// TIA Portal project "DIGITAL ASSEMBLER _Sequential" (V16)
// Vorlageprojekt für das Buch mit Zielsystem S7-1200

(* hardware
DEVICE "S7-1200-Station_1"  S7-1200 Station
   slot 0: "Baugruppenträger_0"  Rack  V1.0
   slot 1: "PLC_1"  CPU 1211C DC/DC/DC  6ES7 211-1AE40-0XB0  V4.1
DEVICE "S7300/ET200M station_1"  S7-300 station
   slot 0: "IO device_1"  IM 153-4 PN  6ES7 153-4BA00-0XB0  V4.0
   slot 0: "Rail_0"  Rail  6ES7 390-1***0-0AA0
   slot 1: "DI 16x24VDC_1"  DI16 x 24VDC  6ES7 321-1BH02-0AA0
   slot 2: "DO 16x24VDC/0.5A_1"  DO16 x 24VDC / 0.5A  6ES7 322-1BH01-0AA0
*)

// ===== PLC "PLC_1"  CPU 1211C DC/DC/DC =====

VAR_GLOBAL   // PLC tag table "Standard-Variablentabelle"
   "counter" AT %QD30 : UDInt;
   "stop light" AT %Q2.3 : Bool;
   "reset light'" AT %Q2.2 : Bool;
   "start light" AT %Q2.1 : Bool;
   "pos rise base" AT %Q2.0 : Bool;
   "clamp base" AT %Q1.7 : Bool;
   "pos rise lid" AT %Q1.6 : Bool;
   "base conveyor" AT %Q1.5 : Bool;
   "clamp lid" AT %Q1.4 : Bool;
   "lids conveyor" AT %Q1.3 : Bool;
   "grab" AT %Q1.2 : Bool;
   "move z" AT %Q1.1 : Bool;
   "move x" AT %Q1.0 : Bool;
   "auto" AT %I2.6 : Bool;
   "emergency stop" AT %I2.5 : Bool;
   "stop" AT %I2.4 : Bool;
   "reset" AT %I2.3 : Bool;
   "start" AT %I2.2 : Bool;
   "part leaving" AT %I2.1 : Bool;
   "pos at limit base" AT %I2.0 : Bool;
   "base clamped" AT %I1.7 : Bool;
   "base at place" AT %I1.6 : Bool;
   "pos at limit lid" AT %I1.5 : Bool;
   "lid clamped" AT %I1.4 : Bool;
   "lid at place" AT %I1.3 : Bool;
   "item detected" AT %I1.2 : Bool;
   "moving z" AT %I1.1 : Bool;
   "moving x" AT %I1.0 : Bool;
   "Manual" AT %I2.7 : Bool;
   "Memory_for_Steps" AT %M0.1 : Bool;
   "Start_FC_one_time" AT %M0.2 : Bool;
   "Tag_1" AT %M0.3 : Bool;
   "Tag_2" AT %M0.4 : Bool;
   "Tag_3" AT %M0.5 : Bool;
   "Tag_4" AT %M0.7 : Bool;
   "Tag_5" AT %M2.7 : Bool;
   "cycle_complete" AT %M3.0 : Bool;
   "Tag_6" AT %M4.1 : Bool;
   "Tag_7" AT %M4.2 : Bool;
   "Tag_8" AT %M5.0 : Bool;
   "Tag_9" AT %M5.1 : Bool;
   "Tag_10" AT %M5.2 : Bool;
   "Tag_11" AT %M5.3 : Bool;
   "Tag_12" AT %M5.4 : Bool;
   "Tag_13" AT %QW30 : Int;
END_VAR

DATA_BLOCK "modes"   // DB1
{ S7_Optimized_Access := 'FALSE' }
VERSION : 0.1
   VAR
      "Reset Mode" : Bool;
      "Manual Mode" : Bool;
      "Auto Mode" : Bool;
   END_VAR
BEGIN
END_DATA_BLOCK

DATA_BLOCK "Step_Data"   // DB2
{ S7_Optimized_Access := 'TRUE' }
VERSION : 0.1
   VAR
      Start_Lids_Conveyor : Bool;   // trun on lids conveyor
      Start_Base_conveyor : Bool;   // turn on base conveyor
      Start_Clamp_Lid : Bool;
      Start_Clamp_Base : Bool;
      Extend_Z_Axis : Bool;
      Extend_x_Axis : Bool;
      Start_Grap : Bool;
      Pose_raise_Base : Bool;
      Every_thing_AT_home : Bool;
   END_VAR
BEGIN
END_DATA_BLOCK

DATA_BLOCK "Steps"   // DB3
{ S7_Optimized_Access := 'TRUE' }
VERSION : 0.1
   VAR
      Current_step : Int;
   END_VAR
BEGIN
END_DATA_BLOCK

// folder: System blocks/Program resources

DATA_BLOCK "IEC_Counter_0_DB"   // DB4
{ S7_Optimized_Access := 'TRUE' }
AUTHOR : Simatic
FAMILY : IEC
NAME : CNTR
VERSION : 1.0
// stored: InstanceOfName IEC_COUNTER
"IEC_COUNTER"
BEGIN
END_DATA_BLOCK

// folder: (top level)

FUNCTION "Operating Mode" : Void   // FC1, LAD
{ S7_Optimized_Access := 'TRUE' }
VERSION : 0.1
   VAR_TEMP   // added for the SCL form of the ladder/FBD networks
      _w1 : Bool;
      _w2 : Bool;
   END_VAR
BEGIN

REGION Network 1
   // manual
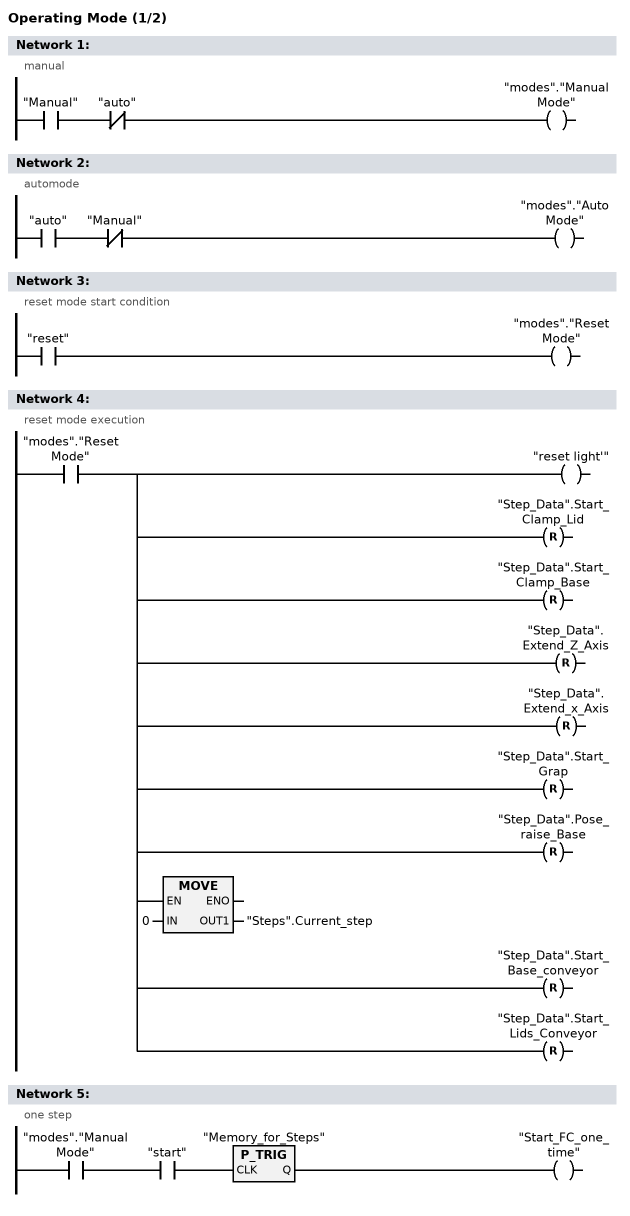
   RUNG wire#powerrail
      Contact( "Manual" )
      I_Contact( "auto" )
      Coil( "modes"."Manual Mode" )
   END_RUNG
   // the same network as SCL:
   "modes"."Manual Mode" := "Manual" AND NOT "auto";
END_REGION

REGION Network 2
   // automode
   RUNG wire#powerrail
      Contact( "auto" )
      I_Contact( "Manual" )
      Coil( "modes"."Auto Mode" )
   END_RUNG
   // the same network as SCL:
   "modes"."Auto Mode" := "auto" AND NOT "Manual";
END_REGION

REGION Network 3
   // reset mode start condition
   RUNG wire#powerrail
      Contact( "reset" )
      Coil( "modes"."Reset Mode" )
   END_RUNG
   // the same network as SCL:
   "modes"."Reset Mode" := "reset";
END_REGION

REGION Network 4
   // reset mode execution
   RUNG wire#powerrail
      Contact( "modes"."Reset Mode" )
      wire#w1
      Coil( "reset light'" )
   END_RUNG
   RUNG wire#w1
      R_Coil( "Step_Data".Start_Clamp_Lid )
   END_RUNG
   RUNG wire#w1
      R_Coil( "Step_Data".Start_Clamp_Base )
   END_RUNG
   RUNG wire#w1
      R_Coil( "Step_Data".Extend_Z_Axis )
   END_RUNG
   RUNG wire#w1
      R_Coil( "Step_Data".Extend_x_Axis )
   END_RUNG
   RUNG wire#w1
      R_Coil( "Step_Data".Start_Grap )
   END_RUNG
   RUNG wire#w1
      R_Coil( "Step_Data".Pose_raise_Base )
   END_RUNG
   RUNG wire#w1
      Move(in := 0, out1 => "Steps".Current_step)
   END_RUNG
   RUNG wire#w1
      R_Coil( "Step_Data".Start_Base_conveyor )
   END_RUNG
   RUNG wire#w1
      R_Coil( "Step_Data".Start_Lids_Conveyor )
   END_RUNG
   // the same network as SCL:
   "reset light'" := "modes"."Reset Mode";
   IF "modes"."Reset Mode" THEN
       "Step_Data".Start_Clamp_Lid := FALSE;
       "Step_Data".Start_Clamp_Base := FALSE;
       "Step_Data".Extend_Z_Axis := FALSE;
       "Step_Data".Extend_x_Axis := FALSE;
       "Step_Data".Start_Grap := FALSE;
       "Step_Data".Pose_raise_Base := FALSE;
       "Steps".Current_step := 0;
       "Step_Data".Start_Base_conveyor := FALSE;
       "Step_Data".Start_Lids_Conveyor := FALSE;
   END_IF;
END_REGION

REGION Network 5
   // one step
   RUNG wire#powerrail
      Contact( "modes"."Manual Mode" )
      Contact( "start" )
      P_Trig( "Memory_for_Steps" )
      Coil( "Start_FC_one_time" )
   END_RUNG
   // the same network as SCL:
   #_w1 := "modes"."Manual Mode" AND "start";
   #_w2 := #_w1 AND NOT "Memory_for_Steps";   // rising edge
   "Memory_for_Steps" := #_w1;
   "Start_FC_one_time" := #_w2;
END_REGION

REGION Network 6
   // make sure envery thing is reseted before starting
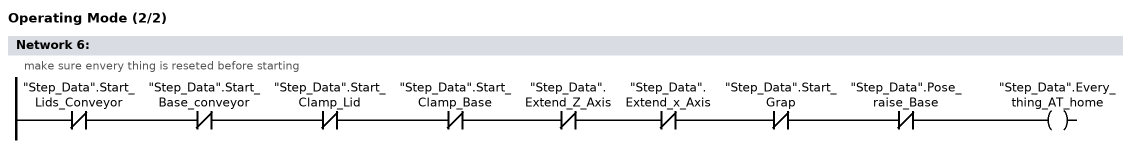
   RUNG wire#powerrail
      I_Contact( "Step_Data".Start_Lids_Conveyor )
      I_Contact( "Step_Data".Start_Base_conveyor )
      I_Contact( "Step_Data".Start_Clamp_Lid )
      I_Contact( "Step_Data".Start_Clamp_Base )
      I_Contact( "Step_Data".Extend_Z_Axis )
      I_Contact( "Step_Data".Extend_x_Axis )
      I_Contact( "Step_Data".Start_Grap )
      I_Contact( "Step_Data".Pose_raise_Base )
      Coil( "Step_Data".Every_thing_AT_home )
   END_RUNG
   // the same network as SCL:
   "Step_Data".Every_thing_AT_home := NOT "Step_Data".Start_Lids_Conveyor AND NOT "Step_Data".Start_Base_conveyor AND NOT "Step_Data".Start_Clamp_Lid AND NOT "Step_Data".Start_Clamp_Base AND NOT "Step_Data".Extend_Z_Axis AND NOT "Step_Data".Extend_x_Axis AND NOT "Step_Data".Start_Grap AND NOT "Step_Data".Pose_raise_Base;
END_REGION
END_FUNCTION

FUNCTION "Step_definition" : Void   // FC2, LAD
{ S7_Optimized_Access := 'TRUE' }
VERSION : 0.1
   VAR_TEMP   // added for the SCL form of the ladder/FBD networks
      _w1 : Bool;
   END_VAR
BEGIN

REGION Network 1: start lids conveyor till lid at place
   // start pressed  and every thing at home
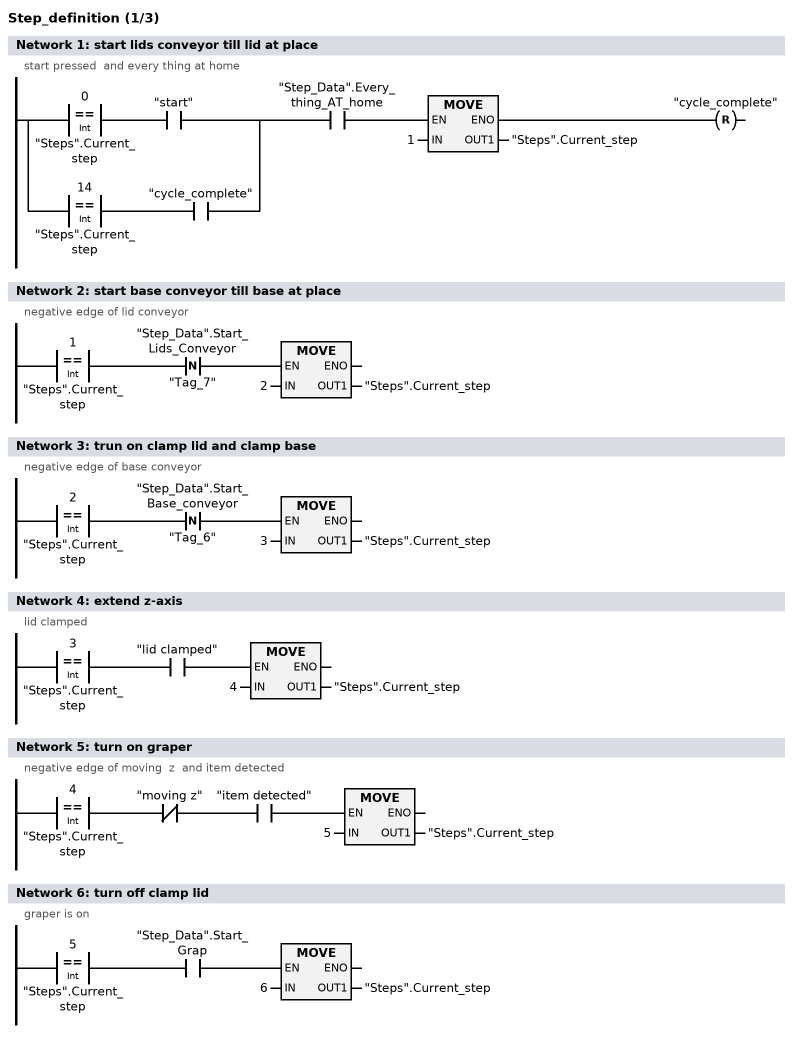
   RUNG wire#powerrail
      { S7_Templates := "SrcType := Int" } EQ_Contact(in1 := 0, in2 := "Steps".Current_step)
      Contact( "start" )
      wire#w1
      Contact( "Step_Data".Every_thing_AT_home )
      Move(in := 1, out1 => "Steps".Current_step)
      R_Coil( "cycle_complete" )
   END_RUNG
   RUNG wire#powerrail
      { S7_Templates := "SrcType := Int" } EQ_Contact(in1 := 14, in2 := "Steps".Current_step)
      Contact( "cycle_complete" )
   END_RUNG wire#w1
   // the same network as SCL:
   #_w1 := (((0 = "Steps".Current_step) AND "start") OR ((14 = "Steps".Current_step) AND "cycle_complete")) AND "Step_Data".Every_thing_AT_home;
   IF #_w1 THEN
       "Steps".Current_step := 1;
       "cycle_complete" := FALSE;
   END_IF;
END_REGION

REGION Network 2: start base conveyor till base at place
   // negative edge of lid conveyor
   RUNG wire#powerrail
      { S7_Templates := "SrcType := Int" } EQ_Contact(in1 := 1, in2 := "Steps".Current_step)
      N_Contact(operand := "Step_Data".Start_Lids_Conveyor, bit := "Tag_7")
      Move(in := 2, out1 => "Steps".Current_step)
   END_RUNG
   // the same network as SCL:
   #_w1 := (1 = "Steps".Current_step) AND NOT "Step_Data".Start_Lids_Conveyor AND "Tag_7";   // falling edge of "Step_Data".Start_Lids_Conveyor
   "Tag_7" := "Step_Data".Start_Lids_Conveyor;
   IF #_w1 THEN "Steps".Current_step := 2; END_IF;
END_REGION

REGION Network 3: trun on clamp lid and clamp base
   // negative edge of base conveyor
   RUNG wire#powerrail
      { S7_Templates := "SrcType := Int" } EQ_Contact(in1 := 2, in2 := "Steps".Current_step)
      N_Contact(operand := "Step_Data".Start_Base_conveyor, bit := "Tag_6")
      Move(in := 3, out1 => "Steps".Current_step)
   END_RUNG
   // the same network as SCL:
   #_w1 := (2 = "Steps".Current_step) AND NOT "Step_Data".Start_Base_conveyor AND "Tag_6";   // falling edge of "Step_Data".Start_Base_conveyor
   "Tag_6" := "Step_Data".Start_Base_conveyor;
   IF #_w1 THEN "Steps".Current_step := 3; END_IF;
END_REGION

REGION Network 4: extend z-axis
   // lid clamped
   RUNG wire#powerrail
      { S7_Templates := "SrcType := Int" } EQ_Contact(in1 := 3, in2 := "Steps".Current_step)
      Contact( "lid clamped" )
      Move(in := 4, out1 => "Steps".Current_step)
   END_RUNG
   // the same network as SCL:
   IF (3 = "Steps".Current_step) AND "lid clamped" THEN "Steps".Current_step := 4; END_IF;
END_REGION

REGION Network 5: turn on graper
   // negative edge of moving  z  and item detected
   RUNG wire#powerrail
      { S7_Templates := "SrcType := Int" } EQ_Contact(in1 := 4, in2 := "Steps".Current_step)
      I_Contact( "moving z" )
      Contact( "item detected" )
      Move(in := 5, out1 => "Steps".Current_step)
   END_RUNG
   // the same network as SCL:
   IF (4 = "Steps".Current_step) AND NOT "moving z" AND "item detected" THEN
       "Steps".Current_step := 5;
   END_IF;
END_REGION

REGION Network 6: turn off clamp lid
   // graper is on
   RUNG wire#powerrail
      { S7_Templates := "SrcType := Int" } EQ_Contact(in1 := 5, in2 := "Steps".Current_step)
      Contact( "Step_Data".Start_Grap )
      Move(in := 6, out1 => "Steps".Current_step)
   END_RUNG
   // the same network as SCL:
   IF (5 = "Steps".Current_step) AND "Step_Data".Start_Grap THEN "Steps".Current_step := 6; END_IF;
END_REGION

REGION Network 7: retract z-axis
   // lid clamped off
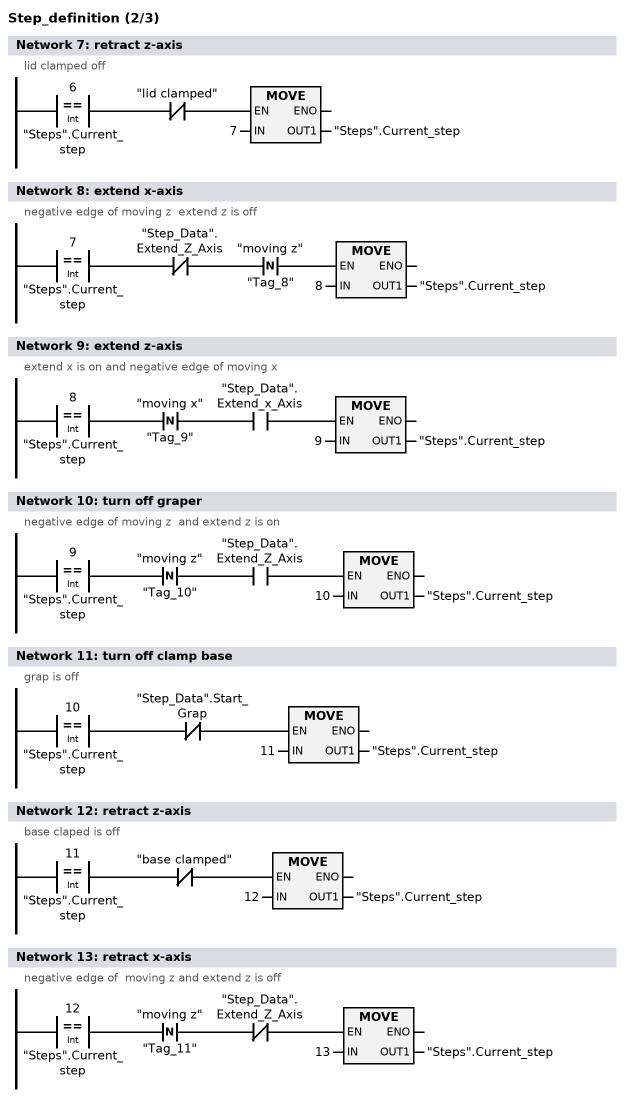
   RUNG wire#powerrail
      { S7_Templates := "SrcType := Int" } EQ_Contact(in1 := 6, in2 := "Steps".Current_step)
      I_Contact( "lid clamped" )
      Move(in := 7, out1 => "Steps".Current_step)
   END_RUNG
   // the same network as SCL:
   IF (6 = "Steps".Current_step) AND NOT "lid clamped" THEN "Steps".Current_step := 7; END_IF;
END_REGION

REGION Network 8: extend x-axis
   // negative edge of moving z  extend z is off
   RUNG wire#powerrail
      { S7_Templates := "SrcType := Int" } EQ_Contact(in1 := 7, in2 := "Steps".Current_step)
      I_Contact( "Step_Data".Extend_Z_Axis )
      N_Contact(operand := "moving z", bit := "Tag_8")
      Move(in := 8, out1 => "Steps".Current_step)
   END_RUNG
   // the same network as SCL:
   #_w1 := (7 = "Steps".Current_step) AND NOT "Step_Data".Extend_Z_Axis AND NOT "moving z" AND "Tag_8";   // falling edge of "moving z"
   "Tag_8" := "moving z";
   IF #_w1 THEN "Steps".Current_step := 8; END_IF;
END_REGION

REGION Network 9: extend z-axis
   // extend x is on and negative edge of moving x
   RUNG wire#powerrail
      { S7_Templates := "SrcType := Int" } EQ_Contact(in1 := 8, in2 := "Steps".Current_step)
      N_Contact(operand := "moving x", bit := "Tag_9")
      Contact( "Step_Data".Extend_x_Axis )
      Move(in := 9, out1 => "Steps".Current_step)
   END_RUNG
   // the same network as SCL:
   #_w1 := (8 = "Steps".Current_step) AND NOT "moving x" AND "Tag_9";   // falling edge of "moving x"
   "Tag_9" := "moving x";
   IF #_w1 AND "Step_Data".Extend_x_Axis THEN "Steps".Current_step := 9; END_IF;
END_REGION

REGION Network 10: turn off graper
   // negative edge of moving z  and extend z is on
   RUNG wire#powerrail
      { S7_Templates := "SrcType := Int" } EQ_Contact(in1 := 9, in2 := "Steps".Current_step)
      N_Contact(operand := "moving z", bit := "Tag_10")
      Contact( "Step_Data".Extend_Z_Axis )
      Move(in := 10, out1 => "Steps".Current_step)
   END_RUNG
   // the same network as SCL:
   #_w1 := (9 = "Steps".Current_step) AND NOT "moving z" AND "Tag_10";   // falling edge of "moving z"
   "Tag_10" := "moving z";
   IF #_w1 AND "Step_Data".Extend_Z_Axis THEN "Steps".Current_step := 10; END_IF;
END_REGION

REGION Network 11: turn off clamp base
   // grap is off
   RUNG wire#powerrail
      { S7_Templates := "SrcType := Int" } EQ_Contact(in1 := 10, in2 := "Steps".Current_step)
      I_Contact( "Step_Data".Start_Grap )
      Move(in := 11, out1 => "Steps".Current_step)
   END_RUNG
   // the same network as SCL:
   IF (10 = "Steps".Current_step) AND NOT "Step_Data".Start_Grap THEN "Steps".Current_step := 11; END_IF;
END_REGION

REGION Network 12: retract z-axis
   // base claped is off
   RUNG wire#powerrail
      { S7_Templates := "SrcType := Int" } EQ_Contact(in1 := 11, in2 := "Steps".Current_step)
      I_Contact( "base clamped" )
      Move(in := 12, out1 => "Steps".Current_step)
   END_RUNG
   // the same network as SCL:
   IF (11 = "Steps".Current_step) AND NOT "base clamped" THEN "Steps".Current_step := 12; END_IF;
END_REGION

REGION Network 13: retract x-axis
   // negative edge of  moving z and extend z is off
   RUNG wire#powerrail
      { S7_Templates := "SrcType := Int" } EQ_Contact(in1 := 12, in2 := "Steps".Current_step)
      N_Contact(operand := "moving z", bit := "Tag_11")
      I_Contact( "Step_Data".Extend_Z_Axis )
      Move(in := 13, out1 => "Steps".Current_step)
   END_RUNG
   // the same network as SCL:
   #_w1 := (12 = "Steps".Current_step) AND NOT "moving z" AND "Tag_11";   // falling edge of "moving z"
   "Tag_11" := "moving z";
   IF #_w1 AND NOT "Step_Data".Extend_Z_Axis THEN "Steps".Current_step := 13; END_IF;
END_REGION

REGION Network 14: pose raise(base on)- base conveyor on till part leaving and counter +1 after part leaving
   // negative edge of  moving x and extend x is off
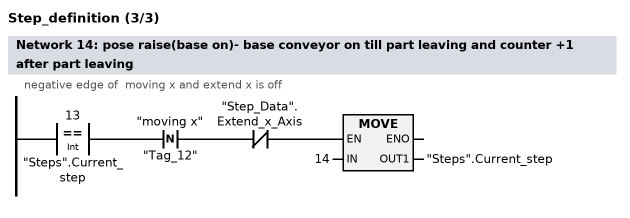
   RUNG wire#powerrail
      { S7_Templates := "SrcType := Int" } EQ_Contact(in1 := 13, in2 := "Steps".Current_step)
      N_Contact(operand := "moving x", bit := "Tag_12")
      I_Contact( "Step_Data".Extend_x_Axis )
      Move(in := 14, out1 => "Steps".Current_step)
   END_RUNG
   // the same network as SCL:
   #_w1 := (13 = "Steps".Current_step) AND NOT "moving x" AND "Tag_12";   // falling edge of "moving x"
   "Tag_12" := "moving x";
   IF #_w1 AND NOT "Step_Data".Extend_x_Axis THEN "Steps".Current_step := 14; END_IF;
END_REGION
END_FUNCTION

FUNCTION "Step_Execution" : Void   // FC3, LAD
{ S7_Optimized_Access := 'TRUE' }
VERSION : 0.1
   VAR_TEMP   // added for the SCL form of the ladder/FBD networks
      _w1 : Bool;
      _w2 : Bool;
   END_VAR
BEGIN

REGION Network 1: trun on lids conveyor
   // start lids conveyor till lid at place
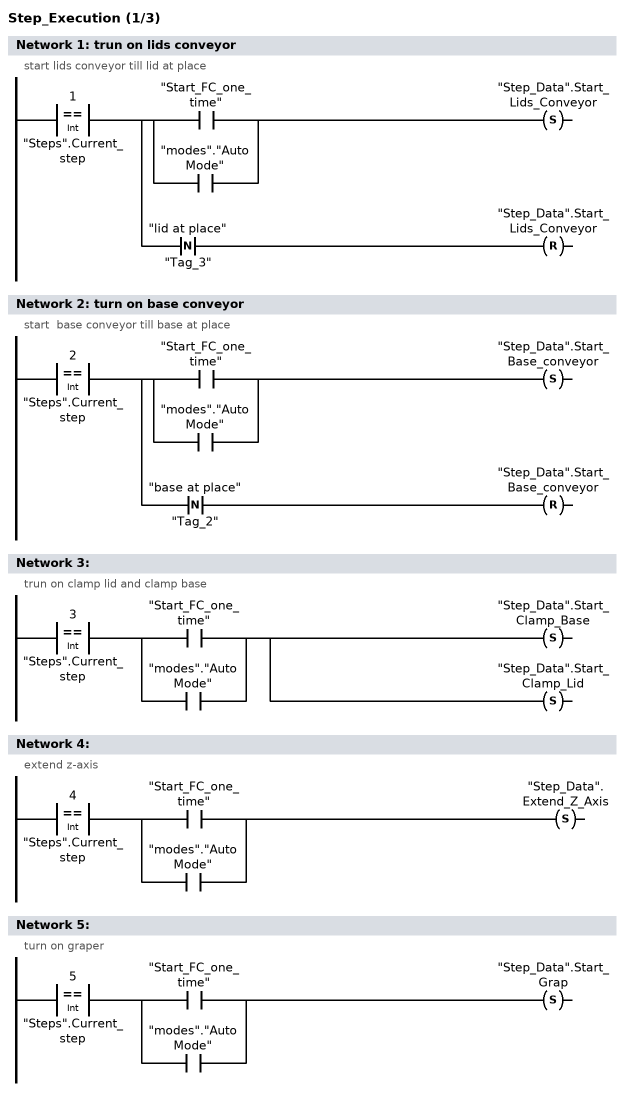
   RUNG wire#powerrail
      { S7_Templates := "SrcType := Int" } EQ_Contact(in1 := 1, in2 := "Steps".Current_step)
      wire#w1
      Contact( "Start_FC_one_time" )
      wire#w2
      S_Coil( "Step_Data".Start_Lids_Conveyor )
   END_RUNG
   RUNG wire#w1
      Contact( "modes"."Auto Mode" )
   END_RUNG wire#w2
   RUNG wire#w1
      N_Contact(operand := "lid at place", bit := "Tag_3")
      R_Coil( "Step_Data".Start_Lids_Conveyor )
   END_RUNG
   // the same network as SCL:
   #_w1 := 1 = "Steps".Current_step;
   IF #_w1 AND ("Start_FC_one_time" OR "modes"."Auto Mode") THEN
       "Step_Data".Start_Lids_Conveyor := TRUE;
   END_IF;
   #_w2 := #_w1 AND NOT "lid at place" AND "Tag_3";   // falling edge of "lid at place"
   "Tag_3" := "lid at place";
   IF #_w2 THEN "Step_Data".Start_Lids_Conveyor := FALSE; END_IF;
END_REGION

REGION Network 2: turn on base conveyor
   // start  base conveyor till base at place
   RUNG wire#powerrail
      { S7_Templates := "SrcType := Int" } EQ_Contact(in1 := 2, in2 := "Steps".Current_step)
      wire#w1
      Contact( "Start_FC_one_time" )
      wire#w2
      S_Coil( "Step_Data".Start_Base_conveyor )
   END_RUNG
   RUNG wire#w1
      Contact( "modes"."Auto Mode" )
   END_RUNG wire#w2
   RUNG wire#w1
      N_Contact(operand := "base at place", bit := "Tag_2")
      R_Coil( "Step_Data".Start_Base_conveyor )
   END_RUNG
   // the same network as SCL:
   #_w1 := 2 = "Steps".Current_step;
   IF #_w1 AND ("Start_FC_one_time" OR "modes"."Auto Mode") THEN
       "Step_Data".Start_Base_conveyor := TRUE;
   END_IF;
   #_w2 := #_w1 AND NOT "base at place" AND "Tag_2";   // falling edge of "base at place"
   "Tag_2" := "base at place";
   IF #_w2 THEN "Step_Data".Start_Base_conveyor := FALSE; END_IF;
END_REGION

REGION Network 3
   // trun on clamp lid and clamp base
   RUNG wire#powerrail
      { S7_Templates := "SrcType := Int" } EQ_Contact(in1 := 3, in2 := "Steps".Current_step)
      wire#w1
      Contact( "Start_FC_one_time" )
      wire#w2
      S_Coil( "Step_Data".Start_Clamp_Base )
   END_RUNG
   RUNG wire#w1
      Contact( "modes"."Auto Mode" )
   END_RUNG wire#w2
   RUNG wire#w2
      S_Coil( "Step_Data".Start_Clamp_Lid )
   END_RUNG
   // the same network as SCL:
   IF (3 = "Steps".Current_step) AND ("Start_FC_one_time" OR "modes"."Auto Mode") THEN
       "Step_Data".Start_Clamp_Base := TRUE;
       "Step_Data".Start_Clamp_Lid := TRUE;
   END_IF;
END_REGION

REGION Network 4
   // extend z-axis
   RUNG wire#powerrail
      { S7_Templates := "SrcType := Int" } EQ_Contact(in1 := 4, in2 := "Steps".Current_step)
      wire#w1
      Contact( "Start_FC_one_time" )
      wire#w2
      S_Coil( "Step_Data".Extend_Z_Axis )
   END_RUNG
   RUNG wire#w1
      Contact( "modes"."Auto Mode" )
   END_RUNG wire#w2
   // the same network as SCL:
   IF (4 = "Steps".Current_step) AND ("Start_FC_one_time" OR "modes"."Auto Mode") THEN
       "Step_Data".Extend_Z_Axis := TRUE;
   END_IF;
END_REGION

REGION Network 5
   // turn on graper
   RUNG wire#powerrail
      { S7_Templates := "SrcType := Int" } EQ_Contact(in1 := 5, in2 := "Steps".Current_step)
      wire#w1
      Contact( "Start_FC_one_time" )
      wire#w2
      S_Coil( "Step_Data".Start_Grap )
   END_RUNG
   RUNG wire#w1
      Contact( "modes"."Auto Mode" )
   END_RUNG wire#w2
   // the same network as SCL:
   IF (5 = "Steps".Current_step) AND ("Start_FC_one_time" OR "modes"."Auto Mode") THEN
       "Step_Data".Start_Grap := TRUE;
   END_IF;
END_REGION

REGION Network 6
   // turn off clamp lid
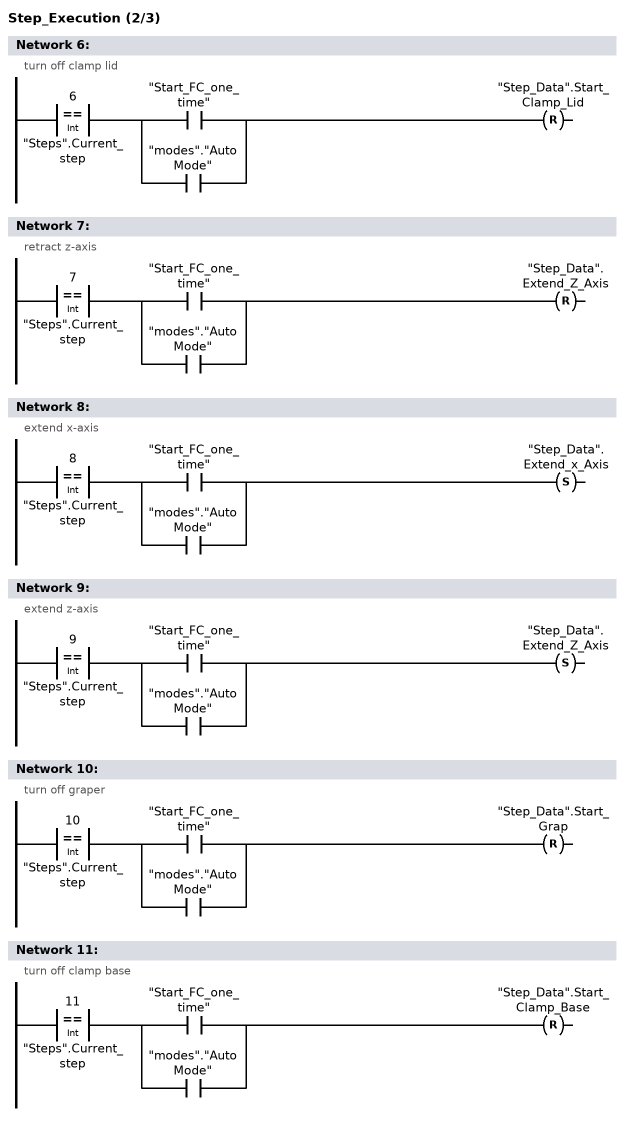
   RUNG wire#powerrail
      { S7_Templates := "SrcType := Int" } EQ_Contact(in1 := 6, in2 := "Steps".Current_step)
      wire#w1
      Contact( "Start_FC_one_time" )
      wire#w2
      R_Coil( "Step_Data".Start_Clamp_Lid )
   END_RUNG
   RUNG wire#w1
      Contact( "modes"."Auto Mode" )
   END_RUNG wire#w2
   // the same network as SCL:
   IF (6 = "Steps".Current_step) AND ("Start_FC_one_time" OR "modes"."Auto Mode") THEN
       "Step_Data".Start_Clamp_Lid := FALSE;
   END_IF;
END_REGION

REGION Network 7
   // retract z-axis
   RUNG wire#powerrail
      { S7_Templates := "SrcType := Int" } EQ_Contact(in1 := 7, in2 := "Steps".Current_step)
      wire#w1
      Contact( "Start_FC_one_time" )
      wire#w2
      R_Coil( "Step_Data".Extend_Z_Axis )
   END_RUNG
   RUNG wire#w1
      Contact( "modes"."Auto Mode" )
   END_RUNG wire#w2
   // the same network as SCL:
   IF (7 = "Steps".Current_step) AND ("Start_FC_one_time" OR "modes"."Auto Mode") THEN
       "Step_Data".Extend_Z_Axis := FALSE;
   END_IF;
END_REGION

REGION Network 8
   // extend x-axis
   RUNG wire#powerrail
      { S7_Templates := "SrcType := Int" } EQ_Contact(in1 := 8, in2 := "Steps".Current_step)
      wire#w1
      Contact( "Start_FC_one_time" )
      wire#w2
      S_Coil( "Step_Data".Extend_x_Axis )
   END_RUNG
   RUNG wire#w1
      Contact( "modes"."Auto Mode" )
   END_RUNG wire#w2
   // the same network as SCL:
   IF (8 = "Steps".Current_step) AND ("Start_FC_one_time" OR "modes"."Auto Mode") THEN
       "Step_Data".Extend_x_Axis := TRUE;
   END_IF;
END_REGION

REGION Network 9
   // extend z-axis
   RUNG wire#powerrail
      { S7_Templates := "SrcType := Int" } EQ_Contact(in1 := 9, in2 := "Steps".Current_step)
      wire#w1
      Contact( "Start_FC_one_time" )
      wire#w2
      S_Coil( "Step_Data".Extend_Z_Axis )
   END_RUNG
   RUNG wire#w1
      Contact( "modes"."Auto Mode" )
   END_RUNG wire#w2
   // the same network as SCL:
   IF (9 = "Steps".Current_step) AND ("Start_FC_one_time" OR "modes"."Auto Mode") THEN
       "Step_Data".Extend_Z_Axis := TRUE;
   END_IF;
END_REGION

REGION Network 10
   // turn off graper
   RUNG wire#powerrail
      { S7_Templates := "SrcType := Int" } EQ_Contact(in1 := 10, in2 := "Steps".Current_step)
      wire#w1
      Contact( "Start_FC_one_time" )
      wire#w2
      R_Coil( "Step_Data".Start_Grap )
   END_RUNG
   RUNG wire#w1
      Contact( "modes"."Auto Mode" )
   END_RUNG wire#w2
   // the same network as SCL:
   IF (10 = "Steps".Current_step) AND ("Start_FC_one_time" OR "modes"."Auto Mode") THEN
       "Step_Data".Start_Grap := FALSE;
   END_IF;
END_REGION

REGION Network 11
   // turn off clamp base
   RUNG wire#powerrail
      { S7_Templates := "SrcType := Int" } EQ_Contact(in1 := 11, in2 := "Steps".Current_step)
      wire#w1
      Contact( "Start_FC_one_time" )
      wire#w2
      R_Coil( "Step_Data".Start_Clamp_Base )
   END_RUNG
   RUNG wire#w1
      Contact( "modes"."Auto Mode" )
   END_RUNG wire#w2
   // the same network as SCL:
   IF (11 = "Steps".Current_step) AND ("Start_FC_one_time" OR "modes"."Auto Mode") THEN
       "Step_Data".Start_Clamp_Base := FALSE;
   END_IF;
END_REGION

REGION Network 12
   // retract z-axis
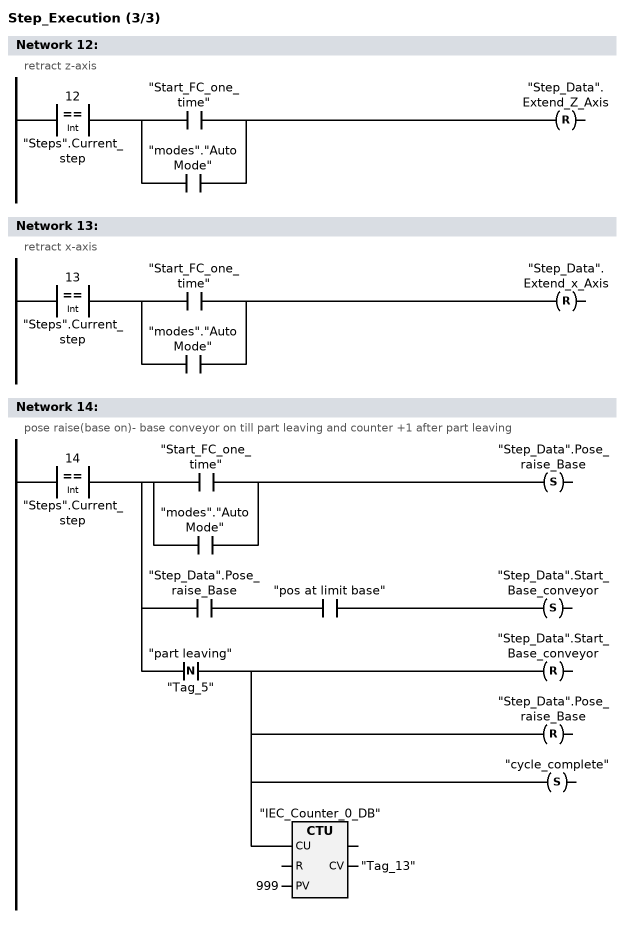
   RUNG wire#powerrail
      { S7_Templates := "SrcType := Int" } EQ_Contact(in1 := 12, in2 := "Steps".Current_step)
      wire#w1
      Contact( "Start_FC_one_time" )
      wire#w2
      R_Coil( "Step_Data".Extend_Z_Axis )
   END_RUNG
   RUNG wire#w1
      Contact( "modes"."Auto Mode" )
   END_RUNG wire#w2
   // the same network as SCL:
   IF (12 = "Steps".Current_step) AND ("Start_FC_one_time" OR "modes"."Auto Mode") THEN
       "Step_Data".Extend_Z_Axis := FALSE;
   END_IF;
END_REGION

REGION Network 13
   // retract x-axis
   RUNG wire#powerrail
      { S7_Templates := "SrcType := Int" } EQ_Contact(in1 := 13, in2 := "Steps".Current_step)
      wire#w1
      Contact( "Start_FC_one_time" )
      wire#w2
      R_Coil( "Step_Data".Extend_x_Axis )
   END_RUNG
   RUNG wire#w1
      Contact( "modes"."Auto Mode" )
   END_RUNG wire#w2
   // the same network as SCL:
   IF (13 = "Steps".Current_step) AND ("Start_FC_one_time" OR "modes"."Auto Mode") THEN
       "Step_Data".Extend_x_Axis := FALSE;
   END_IF;
END_REGION

REGION Network 14
   // pose raise(base on)- base conveyor on till part leaving and counter +1 after part leaving
   #_w1 := 14 = "Steps".Current_step;
   IF #_w1 AND ("Start_FC_one_time" OR "modes"."Auto Mode") THEN "Step_Data".Pose_raise_Base := TRUE; END_IF;
   IF #_w1 AND "Step_Data".Pose_raise_Base AND "pos at limit base" THEN
       "Step_Data".Start_Base_conveyor := TRUE;
   END_IF;
   #_w2 := #_w1 AND NOT "part leaving" AND "Tag_5";   // falling edge of "part leaving"
   "Tag_5" := "part leaving";
   IF #_w2 THEN
       "Step_Data".Start_Base_conveyor := FALSE;
       "Step_Data".Pose_raise_Base := FALSE;
       "cycle_complete" := TRUE;
   END_IF;
   "IEC_Counter_0_DB".CTU(CU := #_w2, PV := 999, CV => "Tag_13");
END_REGION
END_FUNCTION

FUNCTION "Assignment" : Void   // FC4, LAD
{ S7_Optimized_Access := 'TRUE' }
VERSION : 0.1
BEGIN

REGION Network 1
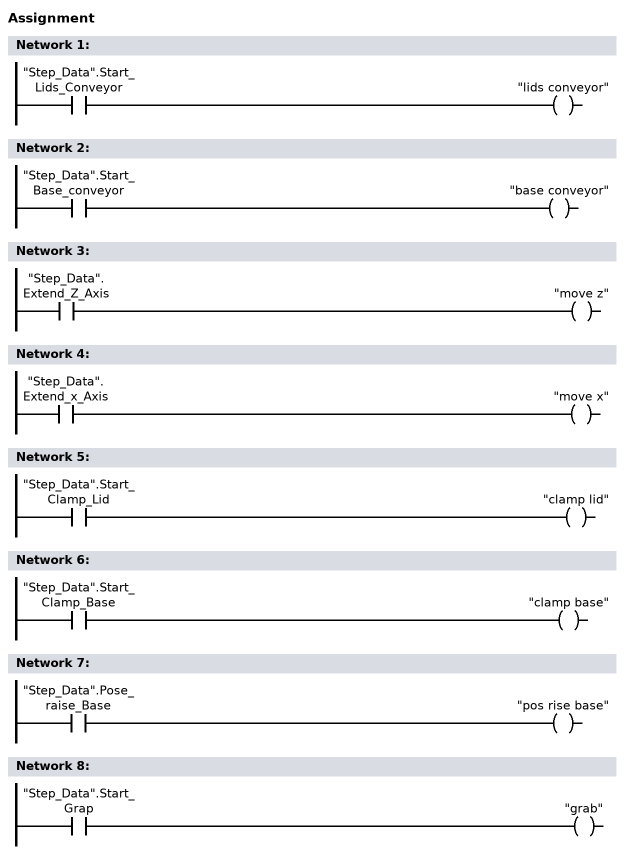
   RUNG wire#powerrail
      Contact( "Step_Data".Start_Lids_Conveyor )
      Coil( "lids conveyor" )
   END_RUNG
   // the same network as SCL:
   "lids conveyor" := "Step_Data".Start_Lids_Conveyor;
END_REGION

REGION Network 2
   RUNG wire#powerrail
      Contact( "Step_Data".Start_Base_conveyor )
      Coil( "base conveyor" )
   END_RUNG
   // the same network as SCL:
   "base conveyor" := "Step_Data".Start_Base_conveyor;
END_REGION

REGION Network 3
   RUNG wire#powerrail
      Contact( "Step_Data".Extend_Z_Axis )
      Coil( "move z" )
   END_RUNG
   // the same network as SCL:
   "move z" := "Step_Data".Extend_Z_Axis;
END_REGION

REGION Network 4
   RUNG wire#powerrail
      Contact( "Step_Data".Extend_x_Axis )
      Coil( "move x" )
   END_RUNG
   // the same network as SCL:
   "move x" := "Step_Data".Extend_x_Axis;
END_REGION

REGION Network 5
   RUNG wire#powerrail
      Contact( "Step_Data".Start_Clamp_Lid )
      Coil( "clamp lid" )
   END_RUNG
   // the same network as SCL:
   "clamp lid" := "Step_Data".Start_Clamp_Lid;
END_REGION

REGION Network 6
   RUNG wire#powerrail
      Contact( "Step_Data".Start_Clamp_Base )
      Coil( "clamp base" )
   END_RUNG
   // the same network as SCL:
   "clamp base" := "Step_Data".Start_Clamp_Base;
END_REGION

REGION Network 7
   RUNG wire#powerrail
      Contact( "Step_Data".Pose_raise_Base )
      Coil( "pos rise base" )
   END_RUNG
   // the same network as SCL:
   "pos rise base" := "Step_Data".Pose_raise_Base;
END_REGION

REGION Network 8
   RUNG wire#powerrail
      Contact( "Step_Data".Start_Grap )
      Coil( "grab" )
   END_RUNG
   // the same network as SCL:
   "grab" := "Step_Data".Start_Grap;
END_REGION
END_FUNCTION

FUNCTION "MHJ-PLC-Lab-Function-S71200" : Void   // FC9000, SCL
{ S7_Optimized_Access := 'TRUE' }
VERSION : 0.1
   VAR_TEMP
      rdTimeReturn : Int;
      outputTime : DTL;
      SyncVal : Byte;
      forVal : Int;
      forVal_2 : Int;
      Value : Byte;
   END_VAR
   VAR CONSTANT
      CompVal : Byte := 16#34;
      Value_01 : Byte := 16#11;
      Value_01_DW : DWord := 16#A165_D992;
      Value_02_DW : DWord := 16#58BE_4401;
   END_VAR
BEGIN

   #Value:=PEEK(area := 16#82,
        dbNumber := 0,
        byteOffset := 511);
   #Value := #Value + 1;

   POKE(area := 16#82,
        dbNumber := 0,
        byteOffset := 511,
        value := #Value);

   POKE(area:=16#81,
        dbNumber:=0,
        byteOffset:=1016,
        value:=#Value_01_DW);
   POKE(area := 16#81,
        dbNumber := 0,
        byteOffset := 1020,
        value := #Value_02_DW);

   POKE(area := 16#81,
        dbNumber := 0,
        byteOffset := 511,
        value := B#16#00);

   FOR #forVal := 0 TO 120 DO
       FOR #forVal_2:=0 TO 10 DO
           #rdTimeReturn:=RD_SYS_T(#outputTime);
           #rdTimeReturn := WR_SYS_T(#outputTime);
           #rdTimeReturn := RD_SYS_T(#outputTime);
           #rdTimeReturn := WR_SYS_T(#outputTime);
       END_FOR;
       #SyncVal:= PEEK(area := 16#81,
                      dbNumber := 0,
                      byteOffset := 511);
       IF #SyncVal = #CompVal THEN
          GOTO M_1;
       END_IF;
   END_FOR;
   RETURN;

   M_1:
   POKE(area := 16#81,
        dbNumber := 0,
        byteOffset := 511,
        value := B#16#0);
END_FUNCTION

ORGANIZATION_BLOCK "Main"   // OB1, LAD, ProgramCycle
TITLE = "Main Program Sweep (Cycle)"
{ S7_Optimized_Access := 'TRUE' }
VERSION : 0.1
   VAR_INPUT
      Initial_Call : Bool;   // Initial call of this OB
      Remanence : Bool;   // =True, if remanent data are available
   END_VAR
BEGIN

REGION Network 1: Konnektierungsbaustein für PLC-Lab
   // Im Netzwerk 1 wird der Konnektierungsbaustein für PLC-Lab aufgerufen.
   // Dieser Aufruf darf nicht entfernt werden!
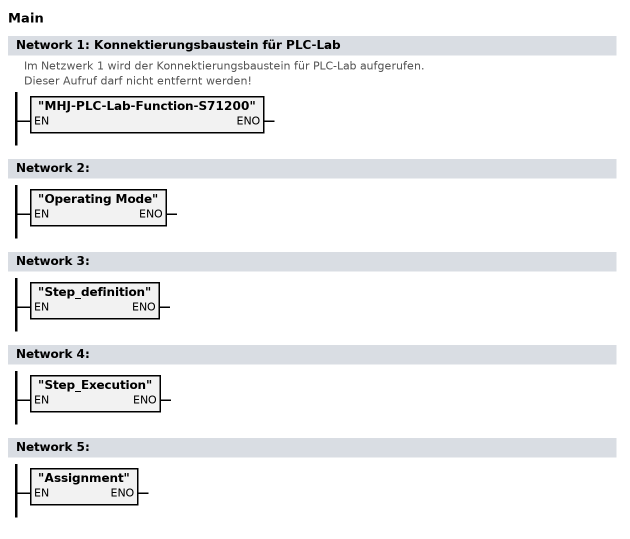
   RUNG wire#powerrail
      "MHJ-PLC-Lab-Function-S71200"()
   END_RUNG
   // the same network as SCL:
   "MHJ-PLC-Lab-Function-S71200"();
END_REGION

REGION Network 2
   RUNG wire#powerrail
      "Operating Mode"()
   END_RUNG
   // the same network as SCL:
   "Operating Mode"();
END_REGION

REGION Network 3
   RUNG wire#powerrail
      "Step_definition"()
   END_RUNG
   // the same network as SCL:
   "Step_definition"();
END_REGION

REGION Network 4
   RUNG wire#powerrail
      "Step_Execution"()
   END_RUNG
   // the same network as SCL:
   "Step_Execution"();
END_REGION

REGION Network 5
   RUNG wire#powerrail
      "Assignment"()
   END_RUNG
   // the same network as SCL:
   "Assignment"();
END_REGION
END_ORGANIZATION_BLOCK